Omron CX-Programmer project 新工程 (CX-Programmer 9.73)

# PLC 新PLC1: CPM1(CPM1A) CPU20

## Global symbols (name address type ; comment)
0.00 BOOL  ; 压力到达
0.02 BOOL  ; 运转准备
0.04 BOOL  ; 不良解除
0.05 BOOL  ; 插头连接好
10.00 BOOL  ; 压力OK
10.01 BOOL  ; BZ
10.02 BOOL  ; NG
10.03 BOOL  ; 放水电磁阀
10.04 BOOL  ; 电机运转
10.05 BOOL  ; 插头检测停止
10.06 BOOL  ; 自动运转中
200.00 BOOL  ; 检查启动PLS
200.01 BOOL  ; 检查中
200.03 BOOL  ; NG不良辅助
200.06 BOOL  ; 检测结束
200.08 BOOL  ; 不良解除辅助
200.09 BOOL  ; 运转准备停止
200.10 BOOL  ; 检测完拔插头提示
201.00 BOOL  ; 拔插头提示
202.00 BOOL  ; 2此检测信号
210.01 BOOL  ; 压力OK辅助
210.02 BOOL  ; 不良提示
CNT000 BOOL  ; 检测次数控制
HR0.00 BOOL  ; STEP1 插头检测断开
HR0.01 BOOL  ; STEP1 水阀开
HR0.01 BOOL  ; STEP2 电机开
HR0.02 BOOL  ; STEP3 电机开
HR0.03 BOOL  ; STEP3 检测等待
HR0.04 BOOL  ; STEP4 电机停
HR0.05 BOOL  ; STEP5 水阀停
HR0.06 BOOL  ; STEP6 检测回路回复
HR0.06 BOOL  ; STEP5 STEP5 水阀停
HR0.07 BOOL  ; STEP7 拔插头提示
HR0.08 BOOL  ; 拔插头等待
HR0.09 BOOL  ; 检测结束
TIM000 BOOL  ; 插头连接确认
TIM001 BOOL  ; 插头拔掉
TIM002 BOOL  ; 插头检测回路断开确认
TIM003 BOOL  ; 放水电磁阀开启延时
TIM005 BOOL  ; 检测等待
TIM006 BOOL  ; 压力到达稳定
TIM007 BOOL  ; 检测结束
TIM008 BOOL  ; 电机运转停止确认
TIM009 BOOL  ; 电机停转检测回路回复
TIM010 BOOL  ; 插头拔掉确认
TIM011 BOOL  ; 拔插头提示时间
TIM012 BOOL  ; 水阀停止确认
TIM018 BOOL  ; 时间长压力到达马上停止

## Program 新程序1 (no task)
; 通过PLC控制器 CPM1(CPM1A) CPU20实现汽车洗涤器电机喷射压力检测模块。 / 系统通过运转准备开关确认生产线就绪后，等待插头连接开关通过插头连接确认定时器确认连接，触发检查启动脉冲，置位检查中标志，点亮自动运转指示灯，开始检测流程。但检查中标志只有在插头连接开关为真、检查中标志未置位且不良指示灯未点亮时才能置位，避免误启动。 / 流程开始后，系统首先进入STEP1 插头检测断开标志，若插头连接开关为假，插头检测回路断开确认定时器计时完成，置位插头检测停止继电器，暂停插头检测。随后，插头检测停止继电器在STEP1 插头检测断开标志置位后保持置位，直到STEP6 检测回路回复标志置位，确保检测过程不受干扰。 / 接着，进入STEP2 水阀开启标志，放水电磁阀开启延时定时器计时完成后打开放水电磁阀，为压力检测提供水流。随后，在STEP3 电机启动标志或STEP3 检测等待标志置位时，若未处于STEP4 电机停止标志、不良辅助标志或2次检测信号状态，启动电机，开始喷射。 / 在STEP3 检测等待标志期间，系统通过检测等待定时器和压力到达稳定定时器监测压力传感器。若计时范围内压力达标，置位压力合格辅助标志，在STEP7 拔插头提示标志置位时点亮压力合格指示灯；若检测结束定时器计时结束仍未达标，置位不良辅助标志，点亮不良指示灯并触发报警蜂鸣器。压力合格辅助标志只有在STEP3 检测等待标志置位且计时范围内压力传感器为真时才能置位，保证压力检测的可靠性。 / 检测完成后，系统进入STEP4 电机停止标志，电机运转停止确认定时器计时完成关闭电机，然后在STEP5 水阀停止标志置位时，水阀停止确认定时器计时完成关闭放水电磁阀。随后，STEP6 检测回路回复标志置位，电机停转检测回路回复定时器计时完成，解除插头检测停止继电器。在STEP7 拔插头提示标志置位时，拔插头提示定时器计时，置位拔插头提示标志提醒操作员拔掉插头。 / 若出现不合格，不良提示标志为真时，操作员需按下不良解除按钮，且不在STEP3 检测等待标志置位时，置位不良解除辅助标志并复位检查中标志，恢复初始状态。不良解除辅助标志只有在不良提示标志为真或系统上电且不在检测等待时才能生效，避免误操作。
Local symbols
不良辅助 200.02 BOOL

### Section 段1

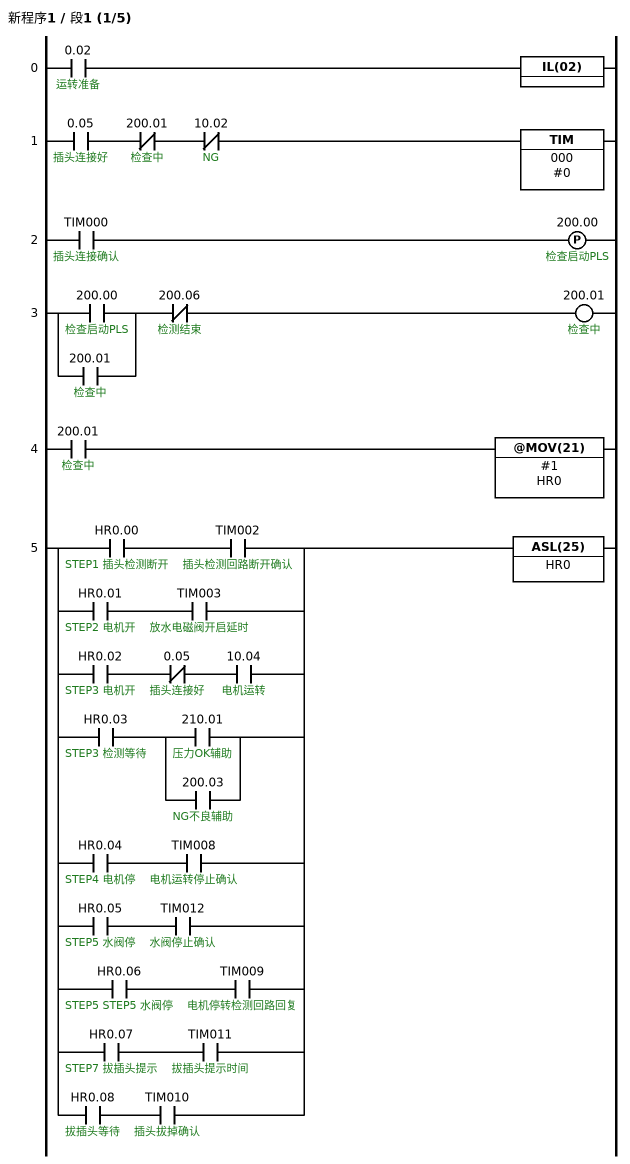
; rung 0
LD 0.02  ; 运转准备
IL(02)
; rung 1
LD 0.05  ; 插头连接好
ANDNOT 200.01  ; 检查中
ANDNOT 10.02  ; NG
TIM 000 #0
; rung 2
LD TIM000  ; 插头连接确认
DIFU(13) 200.00  ; 检查启动PLS
; rung 3
LD 200.00  ; 检查启动PLS
OR 200.01  ; 检查中
ANDNOT 200.06  ; 检测结束
OUT 200.01  ; 检查中
; rung 4
LD 200.01  ; 检查中
@MOV(21) #1 HR0
; rung 5
LD HR0.00  ; STEP1 插头检测断开
AND TIM002  ; 插头检测回路断开确认
LD HR0.01  ; STEP2 电机开
AND TIM003  ; 放水电磁阀开启延时
ORLD
LD HR0.02  ; STEP3 电机开
ANDNOT 0.05  ; 插头连接好
AND 10.04  ; 电机运转
ORLD
LD HR0.03  ; STEP3 检测等待
LD 210.01  ; 压力OK辅助
OR 200.03  ; NG不良辅助
ANDLD
ORLD
LD HR0.04  ; STEP4 电机停
AND TIM008  ; 电机运转停止确认
ORLD
LD HR0.05  ; STEP5 水阀停
AND TIM012  ; 水阀停止确认
ORLD
LD HR0.06  ; STEP5 STEP5 水阀停
AND TIM009  ; 电机停转检测回路回复
ORLD
LD HR0.07  ; STEP7 拔插头提示
AND TIM011  ; 拔插头提示时间
ORLD
LD HR0.08  ; 拔插头等待
AND TIM010  ; 插头拔掉确认
ORLD
ASL(25) HR0

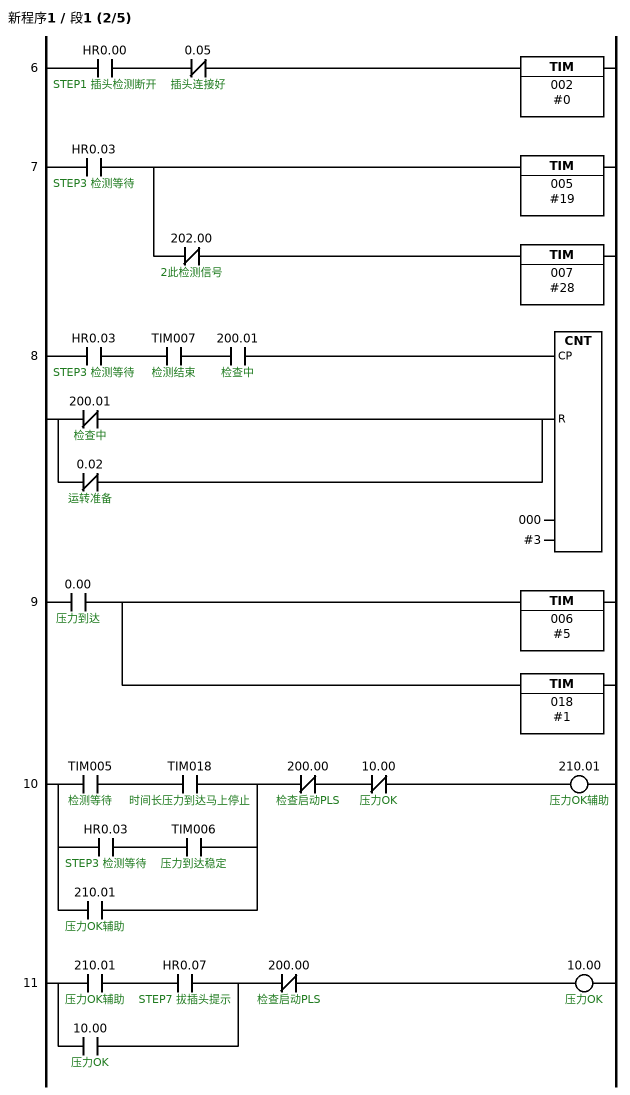
; rung 6
LD HR0.00  ; STEP1 插头检测断开
ANDNOT 0.05  ; 插头连接好
TIM 002 #0
; rung 7
LD HR0.03  ; STEP3 检测等待
TIM 005 #19
ANDNOT 202.00  ; 2此检测信号
TIM 007 #28
; rung 8
LD HR0.03  ; STEP3 检测等待
AND TIM007  ; 检测结束
AND 200.01  ; 检查中
LDNOT 200.01  ; 检查中
ORNOT 0.02  ; 运转准备
CNT 000 #3
; rung 9
LD 0.00  ; 压力到达
TIM 006 #5
TIM 018 #1
; rung 10
LD TIM005  ; 检测等待
AND TIM018  ; 时间长压力到达马上停止
LD HR0.03  ; STEP3 检测等待
AND TIM006  ; 压力到达稳定
ORLD
OR 210.01  ; 压力OK辅助
ANDNOT 200.00  ; 检查启动PLS
ANDNOT 10.00  ; 压力OK
OUT 210.01  ; 压力OK辅助
; rung 11
LD 210.01  ; 压力OK辅助
AND HR0.07  ; STEP7 拔插头提示
OR 10.00  ; 压力OK
ANDNOT 200.00  ; 检查启动PLS
OUT 10.00  ; 压力OK

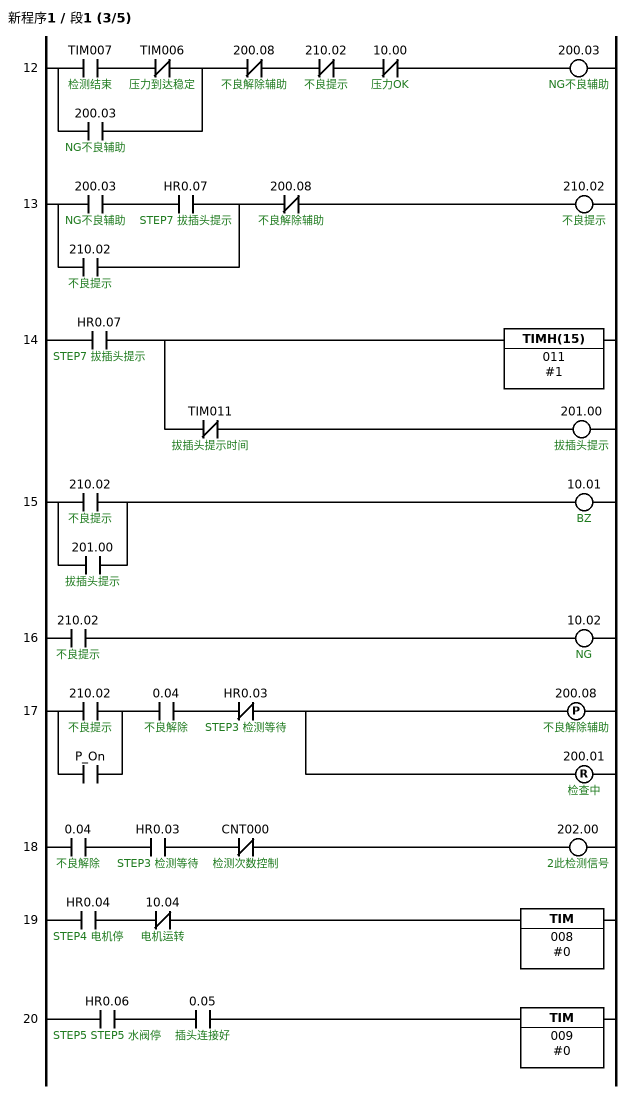
; rung 12
LD TIM007  ; 检测结束
ANDNOT TIM006  ; 压力到达稳定
OR 200.03  ; NG不良辅助
ANDNOT 200.08  ; 不良解除辅助
ANDNOT 210.02  ; 不良提示
ANDNOT 10.00  ; 压力OK
OUT 200.03  ; NG不良辅助
; rung 13
LD 200.03  ; NG不良辅助
AND HR0.07  ; STEP7 拔插头提示
OR 210.02  ; 不良提示
ANDNOT 200.08  ; 不良解除辅助
OUT 210.02  ; 不良提示
; rung 14
LD HR0.07  ; STEP7 拔插头提示
TIMH(15) 011 #1
ANDNOT TIM011  ; 拔插头提示时间
OUT 201.00  ; 拔插头提示
; rung 15
LD 210.02  ; 不良提示
OR 201.00  ; 拔插头提示
OUT 10.01  ; BZ
; rung 16
LD 210.02  ; 不良提示
OUT 10.02  ; NG
; rung 17
LD 210.02  ; 不良提示
OR P_On
AND 0.04  ; 不良解除
ANDNOT HR0.03  ; STEP3 检测等待
DIFU(13) 200.08  ; 不良解除辅助
RSET 200.01  ; 检查中
; rung 18
LD 0.04  ; 不良解除
AND HR0.03  ; STEP3 检测等待
ANDNOT CNT000  ; 检测次数控制
OUT 202.00  ; 2此检测信号
; rung 19
LD HR0.04  ; STEP4 电机停
ANDNOT 10.04  ; 电机运转
TIM 008 #0
; rung 20
LD HR0.06  ; STEP5 STEP5 水阀停
AND 0.05  ; 插头连接好
TIM 009 #0

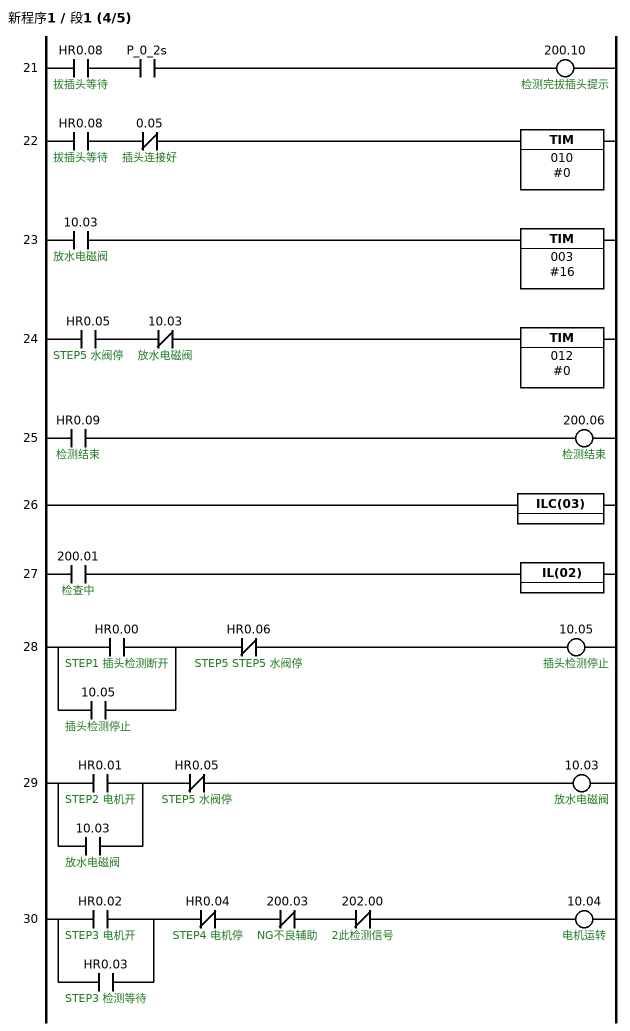
; rung 21
LD HR0.08  ; 拔插头等待
AND P_0_2s
OUT 200.10  ; 检测完拔插头提示
; rung 22
LD HR0.08  ; 拔插头等待
ANDNOT 0.05  ; 插头连接好
TIM 010 #0
; rung 23
LD 10.03  ; 放水电磁阀
TIM 003 #16
; rung 24
LD HR0.05  ; STEP5 水阀停
ANDNOT 10.03  ; 放水电磁阀
TIM 012 #0
; rung 25
LD HR0.09  ; 检测结束
OUT 200.06  ; 检测结束
; rung 26
ILC(03)
; rung 27
LD 200.01  ; 检查中
IL(02)
; rung 28
LD HR0.00  ; STEP1 插头检测断开
OR 10.05  ; 插头检测停止
ANDNOT HR0.06  ; STEP5 STEP5 水阀停
OUT 10.05  ; 插头检测停止
; rung 29
LD HR0.01  ; STEP2 电机开
OR 10.03  ; 放水电磁阀
ANDNOT HR0.05  ; STEP5 水阀停
OUT 10.03  ; 放水电磁阀
; rung 30
LD HR0.02  ; STEP3 电机开
OR HR0.03  ; STEP3 检测等待
ANDNOT HR0.04  ; STEP4 电机停
ANDNOT 200.03  ; NG不良辅助
ANDNOT 202.00  ; 2此检测信号
OUT 10.04  ; 电机运转

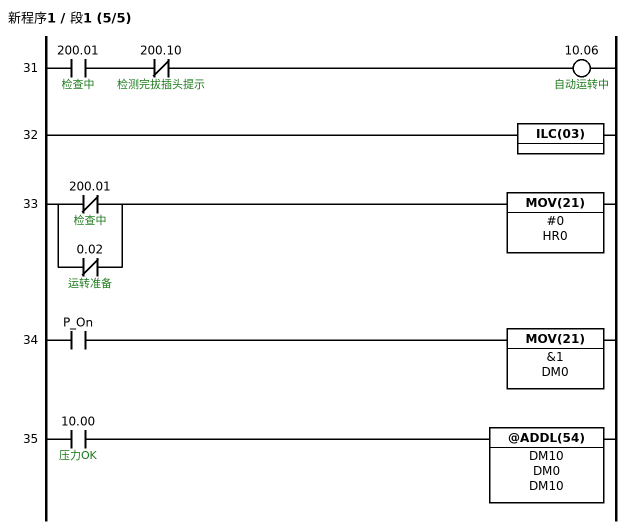
; rung 31
LD 200.01  ; 检查中
ANDNOT 200.10  ; 检测完拔插头提示
OUT 10.06  ; 自动运转中
; rung 32
ILC(03)
; rung 33
LDNOT 200.01  ; 检查中
ORNOT 0.02  ; 运转准备
MOV(21) #0 HR0
; rung 34
LD P_On
MOV(21) &1 DM0
; rung 35
LD 10.00  ; 压力OK
@ADDL(54) DM10 DM0 DM10

### Section END
; rung 0
END(01)